(* IEC 61131-3 sources: IRIS-Project/LASAL CONTROL SOFTWARE/LasalProject_2025_09_12/Class/Manager_Manual_Motor, 1 file *)

(* ---- Manager_Manual_Motor.st ---- *)
(*!
<Class
	Name               = "Manager_Manual_Motor"
	Revision           = "0.0"
	RealtimeTask       = "false"
	CyclicTask         = "true"
	DefCyclictime      = "100 ms"
	BackgroundTask     = "false"
	Sigmatek           = "false"
	OSInterface        = "false"
	HighPriority       = "false"
	Automatic          = "false"
	UpdateMode         = "Prescan"
	SharedCommandTable = "true"
	Objectsize         = "(468,120)">
	<Channels>
		<Server Name="ClassSvr" Visualized="false" Initialize="false" WriteProtected="true" Retentive="false"/>
		<Server Name="S_Mode_Selector" Visualized="false" Initialize="false" WriteProtected="false" Retentive="false"/>
		<Client Name="C_Mode_Selector" Required="false" Internal="false"/>
	</Channels>
</Class>
*)
Manager_Manual_Motor : CLASS
  //Servers:
	ClassSvr 	: SvrChCmd_DINT;
	S_Mode_Selector 	: SvrCh_DINT;
  //Clients:
	C_Mode_Selector 	: CltCh_DINT;
  //Variables:
		v_Mode_selector 	: DINT;
  //Functions:

	FUNCTION VIRTUAL GLOBAL Init;

	FUNCTION VIRTUAL GLOBAL CyWork
		VAR_INPUT
			EAX 	: UDINT;
		END_VAR
		VAR_OUTPUT
			state (EAX) 	: UDINT;
		END_VAR;
  //Tables:
	FUNCTION @STD
		VAR_OUTPUT
			ret_code	: CONFSTATES;
		END_VAR;
	FUNCTION GLOBAL TAB @CT_;
END_CLASS;

FUNCTION VIRTUAL GLOBAL Manager_Manual_Motor::CyWork
	VAR_INPUT
		EAX 	: UDINT;
	END_VAR
	VAR_OUTPUT
		state (EAX) 	: UDINT;
	END_VAR

  if S_Mode_Selector.Read()=1 then
    C_Mode_Selector.Write(input:=1);
  elsif S_Mode_Selector.Read()=0 then
    C_Mode_Selector.Write(input:=0);
  end_if;

	state := READY;

END_FUNCTION

FUNCTION VIRTUAL GLOBAL Manager_Manual_Motor::Init

v_Mode_selector:=0;

END_FUNCTION
